// TIA Portal project "Project1" (V14)

(* hardware
DEVICE "S7-1200 station_1"  S7-1200 Station
   slot 0: "Rack_0"  Rack  V1.0
   slot 1: "PLC_1"  CPU 1211C DC/DC/DC  6ES7 211-1AE40-0XB0  V4.2
DEVICE "PC-System_1"  SIMATIC PC station
   slot 0: "SIMATIC PC station"  Rail  SIMATIC PC-Station  V1.0
      slot 125: "Stationmanager"  Station_Manager  V6.0.4
   slot 1: "HMI_RT_2"  WinCC RT Professional  6AV2 105-0xxxx-xxxx  14.0.0.0
   slot 2: "IE general_1"  IE General  IE_CP  V8.2.0
*)

// ===== PLC "PLC_1"  CPU 1211C DC/DC/DC =====

VAR_GLOBAL   // PLC tag table "Default tag table"
   "Clock_Byte" AT %MB0 : Byte;
   "Clock_10Hz" AT %M0.0 : Bool;
   "Clock_5Hz" AT %M0.1 : Bool;
   "Clock_2.5Hz" AT %M0.2 : Bool;
   "Clock_2Hz" AT %M0.3 : Bool;
   "Clock_1.25Hz" AT %M0.4 : Bool;
   "Clock_1Hz" AT %M0.5 : Bool;
   "Clock_0.625Hz" AT %M0.6 : Bool;
   "Clock_0.5Hz" AT %M0.7 : Bool;
   "System_Byte" AT %MB1 : Byte;
   "FirstScan" AT %M1.0 : Bool;
   "DiagStatusUpdate" AT %M1.1 : Bool;
   "AlwaysTRUE" AT %M1.2 : Bool;
   "AlwaysFALSE" AT %M1.3 : Bool;
END_VAR

ORGANIZATION_BLOCK "Main"   // OB1, LAD, ProgramCycle
TITLE = "Main Program Sweep (Cycle)"
{ S7_Optimized_Access := 'TRUE' }
VERSION : 0.1
   VAR_INPUT
      Initial_Call : Bool;   // Initial call of this OB
      Remanence : Bool;   // =True, if remanent data are available
   END_VAR
BEGIN
END_ORGANIZATION_BLOCK

(* ===== HMI "HMI_RT_2" =====
system functions are stored by id; their names below are inferred from use
connection "HMI_Connection_1": S71200_TCP_IP, SCADA_S7_1200

HMI tags "Default tag table"
   "@HMI_Connection_1@ConnectionState" : DWord AT %DB40000.DBD65000, 500 ms
   "Clock_1Hz" : Bool = PLC Clock_1Hz AT %M0.5, 500 ms
   "@HMI_Connection_1@ForceConnectionState" : DWord AT %DB40000.DBD64000, 500 ms

screen "Screen_1" 1024x768
   Button "Button_1" at 38,338 size 97x31; TextOff 'Stop RT'
      on Click: StopRuntime(0)
   IOField "I/O field_2" at 38,150 size 91x20; FormatPattern FFFFFFFF
      ProcessValue <- "@HMI_Connection_1@ConnectionState"
   IOField "I/O field_3" at 38,93 size 86x20; FormatPattern 1
      ProcessValue <- "Clock_1Hz"
   TextField "Text field_1" at 38,72 size 74x19; Text 'Clock_1Hz'
   TextField "Text field_2" at 38,131 size 279x19; Text '@HMI_Connection_1@ConnectionState'
   IOField "I/O field_1" at 38,223 size 93x20; FormatPattern FFFFFFFF
      ProcessValue <- "@HMI_Connection_1@ConnectionState"
   TextField "Text field_3" at 38,204 size 317x19; Text '@HMI_Connection_1@ForceConnectionState'
   Button "Button_2" at 38,257 size 94x30; TextOff 'Connect'
      on Activate: SetTag("@HMI_Connection_1@ForceConnectionState", 1)
   Button "Button_3" at 38,298 size 96x30; TextOff 'Disconnect'
      on Activate: SetTag("@HMI_Connection_1@ForceConnectionState", 0)
*)